(* PLC project safeApp1, BrAutomation SafeDESIGNER  5.16.0.0 *)
(* stored: companyURL http://www.br-automation.com, creationDateTime Thu Mar 17 10:57:45 2022 *)

PROGRAM Main
  VAR  (* added by the conversion: wires and edge detectors of the diagram *)
    _AND_S68_OUT : ANY;
    _AND_S4_OUT : ANY;
    _BOOL_TO_SAFEBOOL35_OUT : SAFEBOOL;
  END_VAR

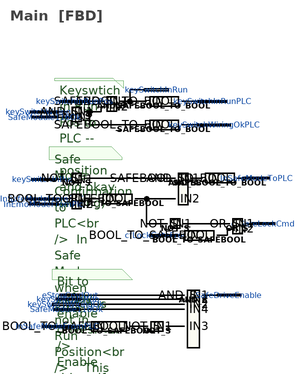
(* FBD diagram, written out as Structured Text *)
(* Keyswtich in Run Pos to PLC -- Needs position and okay (wiring) *)
_AND_S68_OUT := AND_S(keySwitchWiringOk, SafeModule116Ok);
_AND_S4_OUT := AND_S(keySwitchInRunPos, _AND_S68_OUT);
keySwitchInRun := _AND_S4_OUT;
keySwitchInRunPLC := SAFEBOOL_TO_BOOL(_AND_S4_OUT);
keySwitchWiringOkPLC := SAFEBOOL_TO_BOOL(_AND_S68_OUT);
(* Safe Mode Confirmation to PLC<br /> 	In Safe Mode when switch is not in Run Position<br />    This is here in case other logic is needed to confirm safe mode<br /><br />Lock gate when PLC commands it, and not in save mode. *)
_BOOL_TO_SAFEBOOL35_OUT := BOOL_TO_SAFEBOOL(InSafeModeFromPLC OR InEmoModeFromPlc);
InSafeModeToPLC := SAFEBOOL_TO_BOOL(AND_S(NOT_S(keySwitchInRun), _BOOL_TO_SAFEBOOL35_OUT));
cfGateLockCmd := OR_S(NOT_S(_BOOL_TO_SAFEBOOL35_OUT), BOOL_TO_SAFEBOOL(cfLockGateFromPlc));
(* Bit to safely enable drives.<br />    Enable drives if e-stop is okay (high) and not in safe mode (keyswich<br />    or PLC). Consider cutting fluid on an axis by axis basis, so it is easy to <br />    allow some axes to run without the gate closed and locked. *)
SafeDriveEnable := AND_S(eStopCmdOut, keySwitchInRun, keySwitchWiringOk, SafeModule116Ok, NOT_S(BOOL_TO_SAFEBOOL(InSafeModeFromPLC)));
END_PROGRAM
